// Mitsubishi GX Works2 project: 2-input_on.off-belt   PLC: Q02/Q02H

PROGRAM MAIN
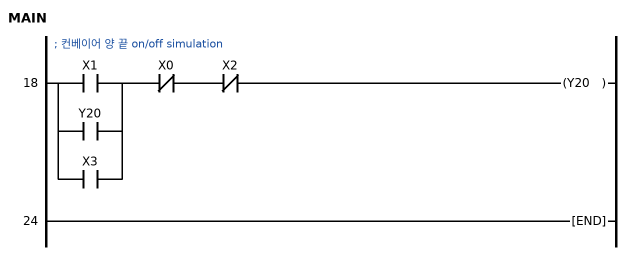
; 컨베이어 양 끝 on/off simulation
18    LD      X1
      OR      Y20
      OR      X3
      ANI     X0
      ANI     X2
      OUT     Y20
24    END
END_PROGRAM
